(* PLC project Relay, NYU-AD Simple 1, author Marios Sazos *)
(* stored: creationDateTime 2017-09-06T16:00:31, version 1, modificationDateTime 2018-04-26T21:54:21 *)

PROGRAM Overcurrent
  VAR
    phase_1 AT %IX0.1 : BOOL;
  END_VAR
  VAR
    trip_fault : BOOL;
  END_VAR
  VAR
    phase_2 AT %IX0.2 : BOOL;
    phase_3 AT %IX0.3 : BOOL;
    local_trip AT %IX0.4 : BOOL;
    local_close AT %IX0.5 : BOOL;
    trip AT %QX0.7 : BOOL;
    close AT %QX0.6 : BOOL;
    remote_trip AT %QX0.0 : BOOL;
    remote_close AT %QX0.1 : BOOL;
    current_RMS AT %MW0 : UINT;
    I_RMS AT %IW0 : UINT;
  END_VAR
  VAR
    T1 : TOF;
    T2 : TON;
    ct_ratio : LINT := 1000;
    current_setpoint : REAL := 500.0;
    a : REAL := 0.02;
    C : REAL := 0.14;
    TMS : REAL := 0.5;
    delay : TIME;
  END_VAR
  VAR
    delay_monitor AT %MW1 : UINT;
  END_VAR
  VAR
    input_pickup : BOOL;
  END_VAR
  VAR  (* added by the conversion: wires and edge detectors of the diagram *)
    _LINT_TO_UINT48_OUT : UINT;
    _UINT_TO_REAL76_OUT : REAL;
    _MUL73_OUT : REAL;
  END_VAR

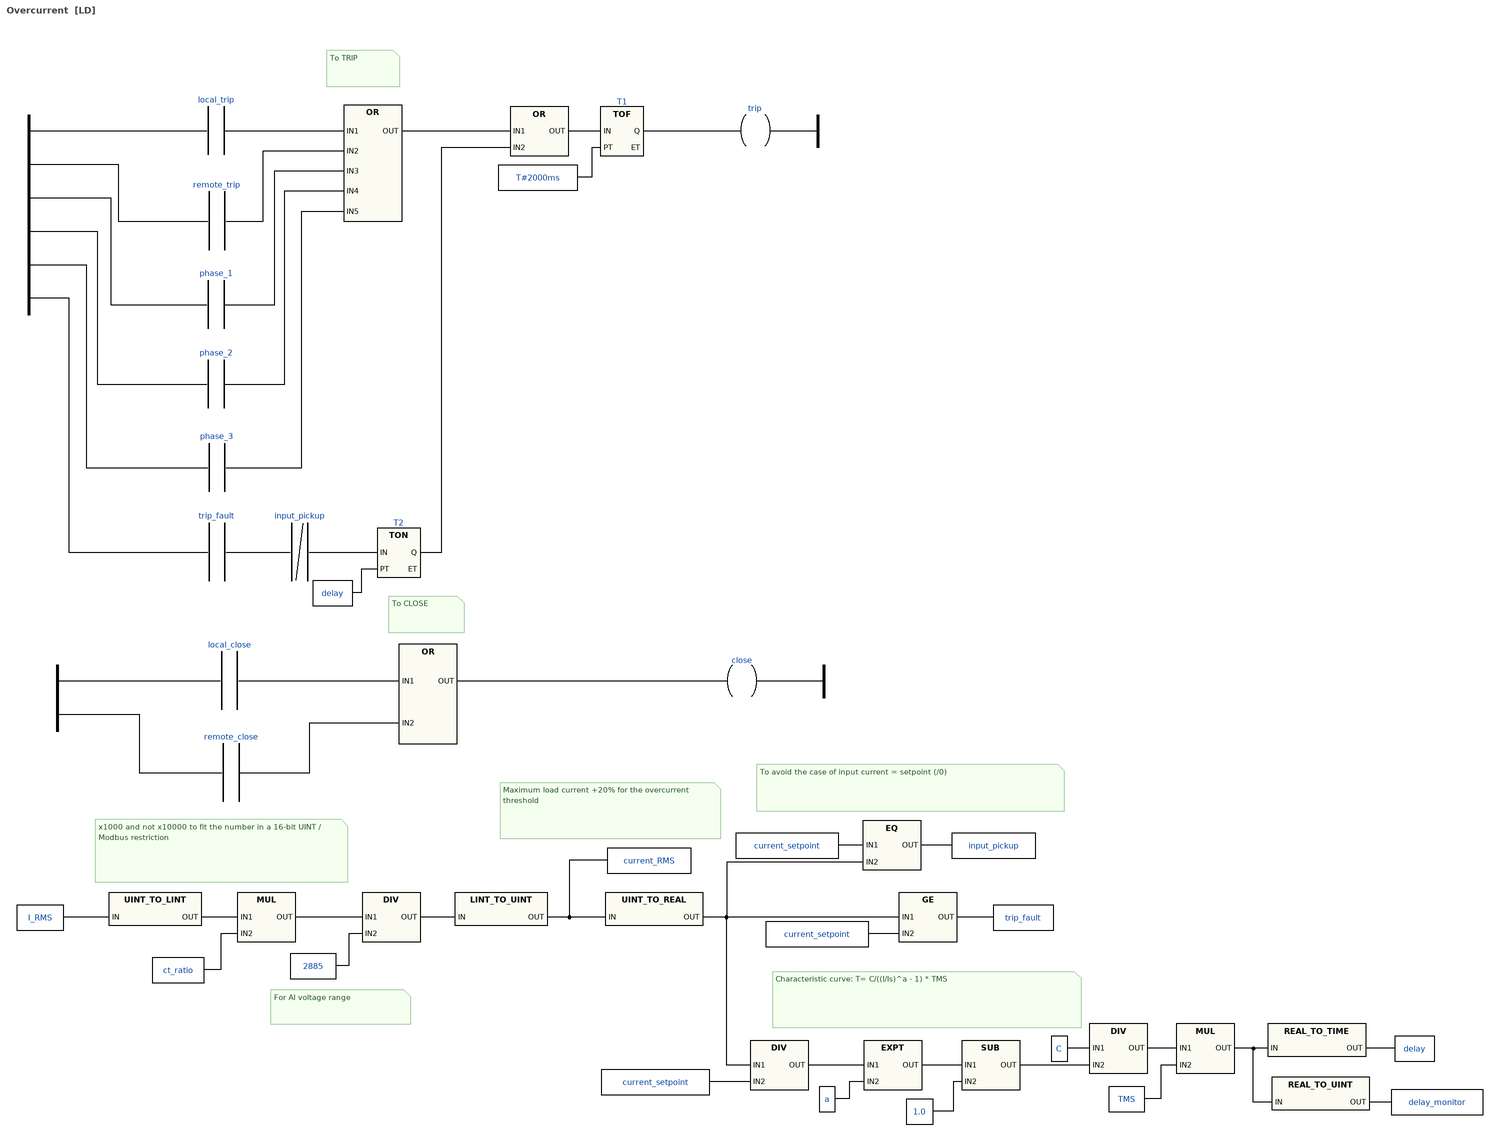
(* LD diagram, written out as Structured Text *)
(* To TRIP *)
T2(IN := trip_fault AND NOT input_pickup, PT := delay);
T1(IN := local_trip OR remote_trip OR phase_1 OR phase_2 OR phase_3 OR T2.Q, PT := T#2000ms);
trip := T1.Q;
(* To CLOSE *)
close := local_close OR remote_close;
(* To avoid the case of input current = setpoint (/0) *)
(* Maximum load current +20% for the overcurrent threshold *)
(* x1000 and not x10000 to fit the number in a 16-bit UINT / Modbus restriction *)
_LINT_TO_UINT48_OUT := LINT_TO_UINT(UINT_TO_LINT(I_RMS) * ct_ratio / 2885);
_UINT_TO_REAL76_OUT := UINT_TO_REAL(_LINT_TO_UINT48_OUT);
input_pickup := current_setpoint = _UINT_TO_REAL76_OUT;
current_RMS := _LINT_TO_UINT48_OUT;
trip_fault := _UINT_TO_REAL76_OUT >= current_setpoint;
(* Characteristic curve: T= C/((I/Is)^a - 1) * TMS *)
(* For AI voltage range *)
_MUL73_OUT := C / (EXPT(_UINT_TO_REAL76_OUT / current_setpoint, a) - 1.0) * TMS;
delay := REAL_TO_TIME(_MUL73_OUT);
delay_monitor := REAL_TO_UINT(_MUL73_OUT);
END_PROGRAM

CONFIGURATION Config0
  RESOURCE Res0 ON PLC
    TASK TaskMain(INTERVAL := T#50ms, PRIORITY := 0);
    PROGRAM Inst0 WITH TaskMain : Overcurrent;
  END_RESOURCE
END_CONFIGURATION
